// Mitsubishi GX Works2 project: 타이머 예제 (무한 반복)   PLC: Q03UDV

PROGRAM MAIN
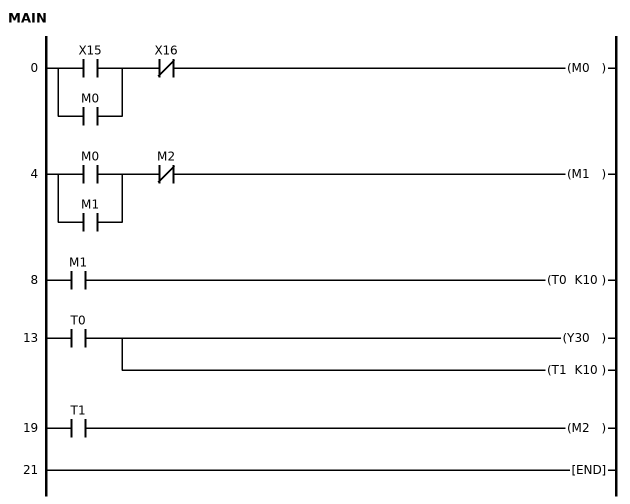
0     LD      X15
      OR      M0
      ANI     X16
      OUT     M0
4     LD      M0
      OR      M1
      ANI     M2
      OUT     M1
8     LD      M1
      OUT     T0 K10
13    LD      T0
      OUT     Y30
      OUT     T1 K10
19    LD      T1
      OUT     M2
21    END
END_PROGRAM
